(* PLC project  *)

CONFIGURATION MainConfig
  VAR_GLOBAL
    GlobalCounter : UDINT;
  END_VAR
  RESOURCE CPU1 ON PLC
    TASK MainTask(INTERVAL := T#10ms, PRIORITY := 1);
    PROGRAM Main : MainProgram;
  END_RESOURCE
END_CONFIGURATION
